PROGRAM GL6_Conveyor
VAR
	GL6_RD: SRoll_Door;
	PASSSED_ROLL_DOOR : BOOL;
	RUN_FWD_BIT_TO_LOAD: BOOL; // RUN FORWARD TO LOAD POSITIONS
	RUN_FWD_BIT_TO_EXIT : BOOL; // RUN FORWARD TO EXIT POSITION AFTER DROP
	JoeBit : BOOL := FALSE;
END_VAR
VAR // added by the converter: edge detectors and wires of the graphical bodies
    _w1 : BOOL;
END_VAR

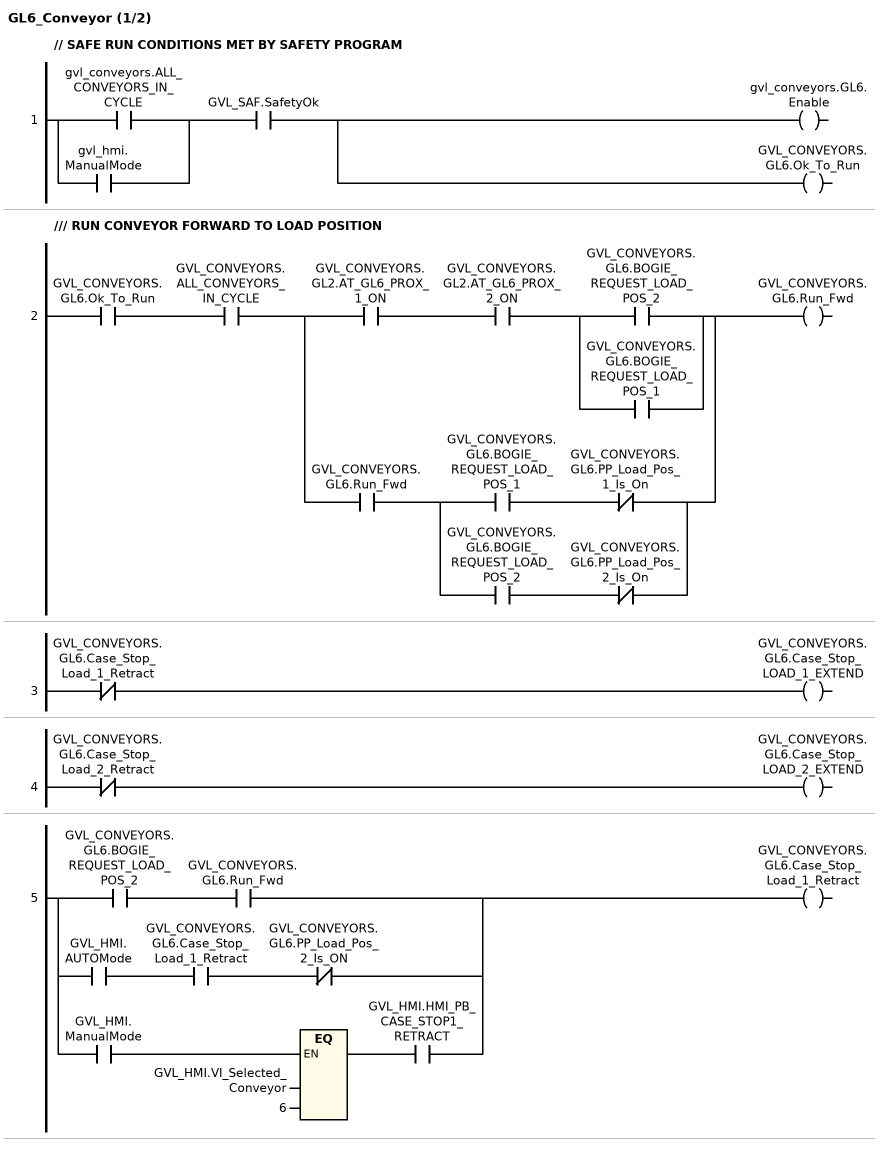
// NETWORK 1: // SAFE RUN CONDITIONS MET BY SAFETY PROGRAM
_w1 := (gvl_conveyors.ALL_CONVEYORS_IN_CYCLE OR gvl_hmi.ManualMode) AND GVL_SAF.SafetyOk;
gvl_conveyors.GL6.Enable := _w1;
GVL_CONVEYORS.GL6.Ok_To_Run := _w1;

// NETWORK 2: /// RUN CONVEYOR FORWARD TO LOAD POSITION
GVL_CONVEYORS.GL6.Run_Fwd := GVL_CONVEYORS.GL6.Ok_To_Run AND GVL_CONVEYORS.ALL_CONVEYORS_IN_CYCLE AND (GVL_CONVEYORS.GL2.AT_GL6_PROX_1_ON AND GVL_CONVEYORS.GL2.AT_GL6_PROX_2_ON AND (GVL_CONVEYORS.GL6.BOGIE_REQUEST_LOAD_POS_2 OR GVL_CONVEYORS.GL6.BOGIE_REQUEST_LOAD_POS_1) OR GVL_CONVEYORS.GL6.Run_Fwd AND (GVL_CONVEYORS.GL6.BOGIE_REQUEST_LOAD_POS_1 AND NOT GVL_CONVEYORS.GL6.PP_Load_Pos_1_Is_On OR GVL_CONVEYORS.GL6.BOGIE_REQUEST_LOAD_POS_2 AND NOT GVL_CONVEYORS.GL6.PP_Load_Pos_2_Is_On));

// NETWORK 3
GVL_CONVEYORS.GL6.Case_Stop_LOAD_1_EXTEND := NOT GVL_CONVEYORS.GL6.Case_Stop_Load_1_Retract;

// NETWORK 4
GVL_CONVEYORS.GL6.Case_Stop_LOAD_2_EXTEND := NOT GVL_CONVEYORS.GL6.Case_Stop_Load_2_Retract;

// NETWORK 5
GVL_CONVEYORS.GL6.Case_Stop_Load_1_Retract := GVL_CONVEYORS.GL6.BOGIE_REQUEST_LOAD_POS_2 AND GVL_CONVEYORS.GL6.Run_Fwd OR GVL_HMI.AUTOMode AND GVL_CONVEYORS.GL6.Case_Stop_Load_1_Retract AND NOT GVL_CONVEYORS.GL6.PP_Load_Pos_2_Is_ON OR (GVL_HMI.ManualMode AND GVL_HMI.VI_Selected_Conveyor = 6) AND GVL_HMI.HMI_PB_CASE_STOP1_RETRACT;

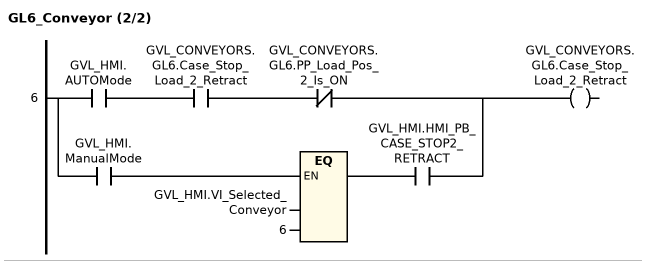
// NETWORK 6
GVL_CONVEYORS.GL6.Case_Stop_Load_2_Retract := GVL_HMI.AUTOMode AND GVL_CONVEYORS.GL6.Case_Stop_Load_2_Retract AND NOT GVL_CONVEYORS.GL6.PP_Load_Pos_2_Is_ON OR (GVL_HMI.ManualMode AND GVL_HMI.VI_Selected_Conveyor = 6) AND GVL_HMI.HMI_PB_CASE_STOP2_RETRACT;

END_PROGRAM

(* stored: Version 1.1.0.1, ProductVersion 3.1.4024.12
   POU GL6_Conveyor: Id {d63fb40f-f7a4-4b7c-ad75-38326a555f6c}, SpecialFunc None *)
